
FUNCTION CB_dint_to_byte : BYTE

TITLE = ' Convert a double integer into a byte '
VERSION : '1.0'
AUTHOR  : CB
NAME    : DintToBy
FAMILY  : TNI

VAR_INPUT
    IN : DINT;
END_VAR

VAR_TEMP

END_VAR

BEGIN

CB_dint_to_byte := DINT_TO_BYTE(IN);

END_FUNCTION
